{attribute addProperty BoxType "EL1918-0000-0016"}
{attribute addProperty Id "Module_1_FSOEModule_1_FSOE_E3D6E7D2104130Module_2_FSLOGICModule_2_FSLOGIC_3E6251391620WcStateAT %I*WcState_98A4DF7520.250InfoDataAT %I*InfoData_BC63D37F80100"}
{attribute addProperty CRC "1996557173"}
{attribute addProperty SizeInBites "202"}
{attribute addProperty SizeInBytes "25.25"}
TYPE EL1918_BB8AB347 :
STRUCT
	{attribute addProperty Name "Module_1_FSOE"}
	Module_1_FSOE : Module_1_FSOE_E3D6E7D2;
	{attribute addProperty Name "Module_2_FSLOGIC"}
	Module_2_FSLOGIC : Module_2_FSLOGIC_3E625139;
	{attribute addProperty Name "WcState"}
	WcState : WcState_98A4DF75;
	{attribute addProperty Name "InfoData"}
	InfoData : InfoData_BC63D37F;
END_STRUCT
END_TYPE

(* stored: Version 1.2.0.0, ProductVersion 3.1.4024.9
   DUT EL1918_BB8AB347: Id {6bcca507-5389-4c46-8e47-06d0917583d1} *)
